PROGRAM MAIN
VAR
END_VAR

END_PROGRAM

(* stored: Version 1.1.0.1
   POU MAIN: Id {cf0ec2f8-d815-47c0-a360-faa36119d775} *)
